FUNCTION_BLOCK CM_ActuatorAnalog
VAR_INPUT
	IN_MANUAL : BOOL;
	IN_AUTO : BOOL;
	IN_HMI_HAND : BOOL;
	
	IN_ON : BOOL;
	IN_OFF : BOOL;
	IN_EMG_STOP : BOOL;
	
	IN_RESET : BOOL;
	
	Input_analog : REAL;
	
	PV : REAL;
END_VAR
VAR_OUTPUT
	HMI_HAND_ON : BOOL;
	output_analog : REAL;
	Output_FB : BOOL;
END_VAR
VAR_IN_OUT
	CM_UDT_CTRL : Udt_CM_ActuatorAnalog;
	Plant_control : Udt_PlantControl;
END_VAR
VAR // added by the converter: edge detectors and wires of the graphical bodies
    _w1 : BOOL;
END_VAR

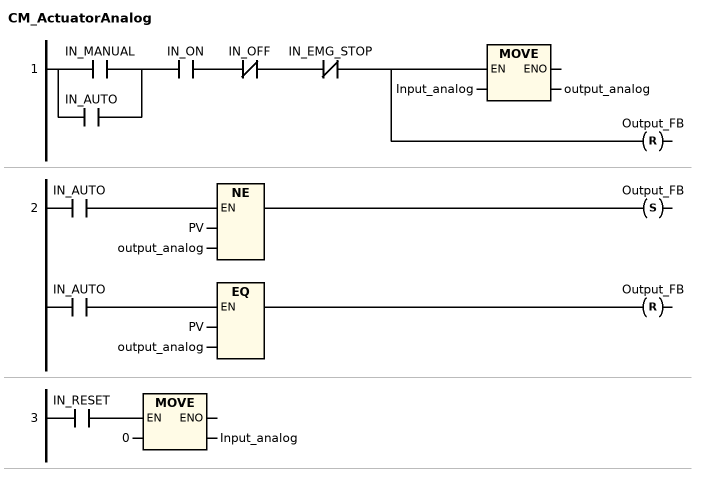
// NETWORK 1
_w1 := (IN_MANUAL OR IN_AUTO) AND IN_ON AND NOT IN_OFF AND NOT IN_EMG_STOP;
IF _w1 THEN output_analog := Input_analog; END_IF
Output_FB R= _w1;

// NETWORK 2
Output_FB S= IN_AUTO AND PV <> output_analog;
Output_FB R= IN_AUTO AND PV = output_analog;

// NETWORK 3
IF IN_RESET THEN Input_analog := 0; END_IF

END_FUNCTION_BLOCK

(* stored: Version 1.1.0.1, ProductVersion 3.1.4024.13
   POU CM_ActuatorAnalog: Id {30afca16-834c-42e1-88e1-c0716c6b03c1}, SpecialFunc None *)
